FUNCTION_BLOCK Q_Priority_AUS (* Command change priority( Part 6 - F.40 ) *)
  (* Standard: ISO 11783-6; Description: Copyright (c) 2022 HR Agrartechnik GmbH This program and the accompanying materials are made available under the terms of the Eclipse Public License 2.0 which is available at https://www.eclipse.org/legal/epl-2.0/ SPDX-License-Identifier: EPL-2.0 see Description Tab *)
  (* Version 1.0, 2025-02-23, Franz Höpfinger, HR Agrartechnik GmbH *)
  PACKAGE isobus::UT::Q;
  IMPORT isobus::UT::Q::const::IDs::ID_NULL;
  (* Documentation:
  Command change priority( Part 6 - F.40 )
   This command is used to change the priority of an alarm mask. This FB wraps isobus::UT::Q::Q_Priority.
   Valid values for u16ObjId (the alarm mask)
   A change-priority Object ID is valid if it falls within the following ISO 11783-6 ID range (Annex F.40):
    - AlarmMask: 2000 – 2999
    ID_NULL (65535) is not a command target but can be used in INIT to deactivate the FB. Any ID outside this range is invalid for commanding.
   param[in] {alarmMaskObjectID, uint16_t}
   Object ID of alarm mask
   param[in] {priority, uint8_t}
   New priority
   Return Values: 
   int16_t
    - VT_E_NO_ERR (0) - OK
   - VT_E_OVERFLOW (-6) - buffer overflow
   - VT_E_NOACT (-8) - Command not possible in current state
   - VT_E_NO_INSTANCE (-21) - No VT client available
   - VT_E_ISO_INSTANCE_INVALID (-129) - Identifier for instance (connection) invalid
   - VT_E_NOT_ALIVE (-130) - Identifier for instance valid, but VT Dead.
  *)
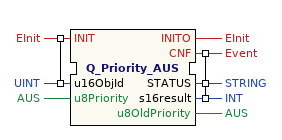
  EVENT_INPUT
    INIT : EInit WITH u16ObjId; (* Service Initialization *)
  END_EVENT
  EVENT_OUTPUT
    INITO : EInit; (* Initialization Confirm *)
    CNF WITH STATUS, s16result; (* Confirmation of Requested Service *)
  END_EVENT
  VAR_INPUT
    u16ObjId : UINT := ID_NULL; (* Object ID *)
  END_VAR
  VAR_OUTPUT
    STATUS : STRING; (* Service Status *)
    s16result : INT; (* retval see description *)
  END_VAR
  SOCKETS
    u8Priority : adapter::types::unidirectional::AUS; (* New priority *)
  END_SOCKETS
  PLUGS
    u8OldPriority : adapter::types::unidirectional::AUS; (* Old priority *)
  END_PLUGS
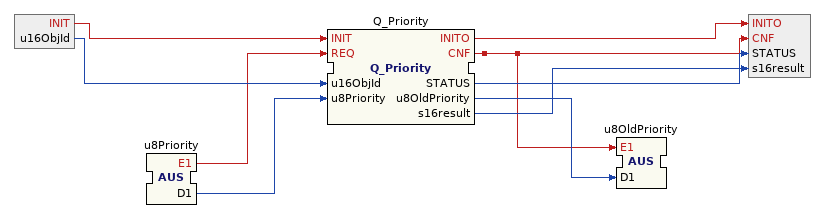
  FBS
    Q_Priority : isobus::UT::Q::Q_Priority;
  END_FBS
  EVENT_CONNECTIONS
    INIT TO Q_Priority.INIT;
    Q_Priority.INITO TO INITO;
    Q_Priority.CNF TO CNF;
    u8Priority.E1 TO Q_Priority.REQ;
    Q_Priority.CNF TO u8OldPriority.E1;
  END_CONNECTIONS
  DATA_CONNECTIONS
    Q_Priority.STATUS TO STATUS;
    u16ObjId TO Q_Priority.u16ObjId;
    u8Priority.D1 TO Q_Priority.u8Priority;
    Q_Priority.u8OldPriority TO u8OldPriority.D1;
    Q_Priority.s16result TO s16result;
  END_CONNECTIONS
END_FUNCTION_BLOCK
